{attribute addProperty BoxType "EK1100-0000-0018"}
{attribute addProperty Id "Beckhoff_EL32xxEK1122Beckhoff_EL32xxEK1122_91C4062C162A_0001_EL3201_0000_0016EL3201_E6230DF016821A_0002_EL3201_0000_0017EL3201_D2AFA85617722.125A_0003_EL3201_0000_0018EL3201_D2AFA85617722.125A_0004_EL3201_0000_0019EL3201_D2AFA85617722.125A_0005_EL3201_0000_0020EL3201_D2AFA85617722.125A_0006_EL3201_0000_0021EL3201_D2AFA85617722.125A_0007_EL3201_0000_0022EL3201_D2AFA85617722.125A_0008_EL3201_0010_0016EL3201_E6230DF016821A_0009_EL3201_0010_0017EL3201_D2AFA85617722.125A_0010_EL3201_0010_0018EL3201_D2AFA85617722.125A_0011_EL3201_0010_0019EL3201_D2AFA85617722.125A_0012_EL3201_0010_0020EL3201_D2AFA85617722.125A_0013_EL3201_0010_0021EL3201_D2AFA85617722.125A_0014_EL3201_0010_0022EL3201_D2AFA85617722.125A_0015_EL3201_0020_0016EL3201_E6230DF016821A_0016_EL3201_0020_0017EL3201_D2AFA85617722.125A_0017_EL3201_0020_0018EL3201_D2AFA85617722.125A_0018_EL3201_0020_0019EL3201_D2AFA85617722.125A_0019_EL3201_0020_0020EL3201_D2AFA85617722.125A_0020_EL3201_0020_0021EL3201_D2AFA85617722.125A_0021_EL3201_0020_0022EL3201_D2AFA85617722.125A_0022_EL3202_0000_0016EL3202_DE79C1A224030A_0023_EL3202_0000_0017EL3202_5359D6C325832.25A_0024_EL3202_0000_0018EL3202_5359D6C325832.25A_0025_EL3202_0000_0019EL3202_5359D6C325832.25A_0026_EL3202_0000_0020EL3202_5359D6C325832.25A_0027_EL3202_0000_0021EL3202_5359D6C325832.25A_0028_EL3202_0000_0022EL3202_5359D6C325832.25A_0029_EL3202_0010_0016EL3202_DE79C1A224030A_0030_EL3202_0010_0017EL3202_5359D6C325832.25A_0031_EL3202_0010_0018EL3202_5359D6C325832.25A_0032_EL3202_0010_0019EL3202_5359D6C325832.25A_0033_EL3202_0010_0020EL3202_5359D6C325832.25A_0034_EL3202_0010_0021EL3202_5359D6C325832.25A_0035_EL3202_0010_0022EL3202_5359D6C325832.25A_0036_EL3202_0020_0017EL3202_5359D6C325832.25A_0037_EL3202_0020_0018EL3202_5359D6C325832.25A_0038_EL3202_0020_0019EL3202_5359D6C325832.25A_0039_EL3202_0020_0020EL3202_5359D6C325832.25A_0040_EL3202_0020_0021EL3202_5359D6C325832.25A_0041_EL3202_0020_0022EL3202_5359D6C325832.25A_0042_EL3204_0000_0016EL3204_5D3AF62938448A_0043_EL3204_0000_0017EL3204_6E5DE15842052.5A_0044_EL3204_0000_0018EL3204_6E5DE15842052.5A_0045_EL3204_0000_0019EL3204_6E5DE15842052.5A_0046_EL3204_0000_0020EL3204_6E5DE15842052.5A_0047_EL3204_0000_0021EL3204_6E5DE15842052.5A_0048_EL3204_0162_0016EL3204_34C8240A22428A_0049_EL3204_0162_0017EL3204_34C8240A22428A_0050_EL3204_0162_0018EL3204_34C8240A22428A_0051_EL3204_0162_0019EL3204_34C8240A22428A_0052_EL3204_0200_0016EL3204_6BC1D0AA22428A_0053_EL3204_0200_0017EL3204_6BC1D0AA22428A_0054_EL3204_0200_0018EL3204_6BC1D0AA22428A_0055_EL3208_0000_0017EL3208_6C7FE11635244A_0056_EL3208_0000_0018EL3208_6C7FE11635244A_0057_EL3208_0010_0016EL3208_6C7FE11635244A_0058_EL3214_0000_0016EL3214_6BC1D0AA22428A_0059_EL3214_0000_0017EL3214_6BC1D0AA22428A_0060_EL3214_0090_0016EL3214_6BC1D0AA22428A_0061_EL3218_0000_0016EL3218_6C7FE11635244A_0062_EL3218_0000_0017EL3218_6C7FE11635244A_0063_EL3255_0000_0016EL3255_3E81353E25632A_0064_EL3255_0000_0017EL3255_0AEBB40125632A_0065_EL3255_0000_0018EL3255_0AEBB40125632A_0066_EL3255_0000_0019EL3255_0AEBB40125632A_0067_EL3255_0000_0020EL3255_2CD3FD4820826A_0068_EL3255_0000_0021EL3255_A08AFE1A25632A_0069_EL3255_0000_0022EL3255_A08AFE1A25632A_0070_EL3255_0000_0023EL3255_A08AFE1A25632"}
{attribute addProperty CRC "491847296"}
{attribute addProperty SizeInBites "17314"}
{attribute addProperty SizeInBytes "2164.25"}
TYPE Beckhoff_EL32xx_1D50FE80 EXTENDS EK1100_179A0949 :
STRUCT
	{attribute addProperty Name "Beckhoff_EL32xxEK1122"}
	Beckhoff_EL32xxEK1122 : Beckhoff_EL32xxEK1122_91C4062C;
	{attribute addProperty Name "A_0001_EL3201_0000_0016"}
	A_0001_EL3201_0000_0016 : EL3201_E6230DF0;
	{attribute addProperty Name "A_0002_EL3201_0000_0017"}
	A_0002_EL3201_0000_0017 : EL3201_D2AFA856;
	{attribute addProperty Name "A_0003_EL3201_0000_0018"}
	A_0003_EL3201_0000_0018 : EL3201_D2AFA856;
	{attribute addProperty Name "A_0004_EL3201_0000_0019"}
	A_0004_EL3201_0000_0019 : EL3201_D2AFA856;
	{attribute addProperty Name "A_0005_EL3201_0000_0020"}
	A_0005_EL3201_0000_0020 : EL3201_D2AFA856;
	{attribute addProperty Name "A_0006_EL3201_0000_0021"}
	A_0006_EL3201_0000_0021 : EL3201_D2AFA856;
	{attribute addProperty Name "A_0007_EL3201_0000_0022"}
	A_0007_EL3201_0000_0022 : EL3201_D2AFA856;
	{attribute addProperty Name "A_0008_EL3201_0010_0016"}
	A_0008_EL3201_0010_0016 : EL3201_E6230DF0;
	{attribute addProperty Name "A_0009_EL3201_0010_0017"}
	A_0009_EL3201_0010_0017 : EL3201_D2AFA856;
	{attribute addProperty Name "A_0010_EL3201_0010_0018"}
	A_0010_EL3201_0010_0018 : EL3201_D2AFA856;
	{attribute addProperty Name "A_0011_EL3201_0010_0019"}
	A_0011_EL3201_0010_0019 : EL3201_D2AFA856;
	{attribute addProperty Name "A_0012_EL3201_0010_0020"}
	A_0012_EL3201_0010_0020 : EL3201_D2AFA856;
	{attribute addProperty Name "A_0013_EL3201_0010_0021"}
	A_0013_EL3201_0010_0021 : EL3201_D2AFA856;
	{attribute addProperty Name "A_0014_EL3201_0010_0022"}
	A_0014_EL3201_0010_0022 : EL3201_D2AFA856;
	{attribute addProperty Name "A_0015_EL3201_0020_0016"}
	A_0015_EL3201_0020_0016 : EL3201_E6230DF0;
	{attribute addProperty Name "A_0016_EL3201_0020_0017"}
	A_0016_EL3201_0020_0017 : EL3201_D2AFA856;
	{attribute addProperty Name "A_0017_EL3201_0020_0018"}
	A_0017_EL3201_0020_0018 : EL3201_D2AFA856;
	{attribute addProperty Name "A_0018_EL3201_0020_0019"}
	A_0018_EL3201_0020_0019 : EL3201_D2AFA856;
	{attribute addProperty Name "A_0019_EL3201_0020_0020"}
	A_0019_EL3201_0020_0020 : EL3201_D2AFA856;
	{attribute addProperty Name "A_0020_EL3201_0020_0021"}
	A_0020_EL3201_0020_0021 : EL3201_D2AFA856;
	{attribute addProperty Name "A_0021_EL3201_0020_0022"}
	A_0021_EL3201_0020_0022 : EL3201_D2AFA856;
	{attribute addProperty Name "A_0022_EL3202_0000_0016"}
	A_0022_EL3202_0000_0016 : EL3202_DE79C1A2;
	{attribute addProperty Name "A_0023_EL3202_0000_0017"}
	A_0023_EL3202_0000_0017 : EL3202_5359D6C3;
	{attribute addProperty Name "A_0024_EL3202_0000_0018"}
	A_0024_EL3202_0000_0018 : EL3202_5359D6C3;
	{attribute addProperty Name "A_0025_EL3202_0000_0019"}
	A_0025_EL3202_0000_0019 : EL3202_5359D6C3;
	{attribute addProperty Name "A_0026_EL3202_0000_0020"}
	A_0026_EL3202_0000_0020 : EL3202_5359D6C3;
	{attribute addProperty Name "A_0027_EL3202_0000_0021"}
	A_0027_EL3202_0000_0021 : EL3202_5359D6C3;
	{attribute addProperty Name "A_0028_EL3202_0000_0022"}
	A_0028_EL3202_0000_0022 : EL3202_5359D6C3;
	{attribute addProperty Name "A_0029_EL3202_0010_0016"}
	A_0029_EL3202_0010_0016 : EL3202_DE79C1A2;
	{attribute addProperty Name "A_0030_EL3202_0010_0017"}
	A_0030_EL3202_0010_0017 : EL3202_5359D6C3;
	{attribute addProperty Name "A_0031_EL3202_0010_0018"}
	A_0031_EL3202_0010_0018 : EL3202_5359D6C3;
	{attribute addProperty Name "A_0032_EL3202_0010_0019"}
	A_0032_EL3202_0010_0019 : EL3202_5359D6C3;
	{attribute addProperty Name "A_0033_EL3202_0010_0020"}
	A_0033_EL3202_0010_0020 : EL3202_5359D6C3;
	{attribute addProperty Name "A_0034_EL3202_0010_0021"}
	A_0034_EL3202_0010_0021 : EL3202_5359D6C3;
	{attribute addProperty Name "A_0035_EL3202_0010_0022"}
	A_0035_EL3202_0010_0022 : EL3202_5359D6C3;
	{attribute addProperty Name "A_0036_EL3202_0020_0017"}
	A_0036_EL3202_0020_0017 : EL3202_5359D6C3;
	{attribute addProperty Name "A_0037_EL3202_0020_0018"}
	A_0037_EL3202_0020_0018 : EL3202_5359D6C3;
	{attribute addProperty Name "A_0038_EL3202_0020_0019"}
	A_0038_EL3202_0020_0019 : EL3202_5359D6C3;
	{attribute addProperty Name "A_0039_EL3202_0020_0020"}
	A_0039_EL3202_0020_0020 : EL3202_5359D6C3;
	{attribute addProperty Name "A_0040_EL3202_0020_0021"}
	A_0040_EL3202_0020_0021 : EL3202_5359D6C3;
	{attribute addProperty Name "A_0041_EL3202_0020_0022"}
	A_0041_EL3202_0020_0022 : EL3202_5359D6C3;
	{attribute addProperty Name "A_0042_EL3204_0000_0016"}
	A_0042_EL3204_0000_0016 : EL3204_5D3AF629;
	{attribute addProperty Name "A_0043_EL3204_0000_0017"}
	A_0043_EL3204_0000_0017 : EL3204_6E5DE158;
	{attribute addProperty Name "A_0044_EL3204_0000_0018"}
	A_0044_EL3204_0000_0018 : EL3204_6E5DE158;
	{attribute addProperty Name "A_0045_EL3204_0000_0019"}
	A_0045_EL3204_0000_0019 : EL3204_6E5DE158;
	{attribute addProperty Name "A_0046_EL3204_0000_0020"}
	A_0046_EL3204_0000_0020 : EL3204_6E5DE158;
	{attribute addProperty Name "A_0047_EL3204_0000_0021"}
	A_0047_EL3204_0000_0021 : EL3204_6E5DE158;
	{attribute addProperty Name "A_0048_EL3204_0162_0016"}
	A_0048_EL3204_0162_0016 : EL3204_34C8240A;
	{attribute addProperty Name "A_0049_EL3204_0162_0017"}
	A_0049_EL3204_0162_0017 : EL3204_34C8240A;
	{attribute addProperty Name "A_0050_EL3204_0162_0018"}
	A_0050_EL3204_0162_0018 : EL3204_34C8240A;
	{attribute addProperty Name "A_0051_EL3204_0162_0019"}
	A_0051_EL3204_0162_0019 : EL3204_34C8240A;
	{attribute addProperty Name "A_0052_EL3204_0200_0016"}
	A_0052_EL3204_0200_0016 : EL3204_6BC1D0AA;
	{attribute addProperty Name "A_0053_EL3204_0200_0017"}
	A_0053_EL3204_0200_0017 : EL3204_6BC1D0AA;
	{attribute addProperty Name "A_0054_EL3204_0200_0018"}
	A_0054_EL3204_0200_0018 : EL3204_6BC1D0AA;
	{attribute addProperty Name "A_0055_EL3208_0000_0017"}
	A_0055_EL3208_0000_0017 : EL3208_6C7FE116;
	{attribute addProperty Name "A_0056_EL3208_0000_0018"}
	A_0056_EL3208_0000_0018 : EL3208_6C7FE116;
	{attribute addProperty Name "A_0057_EL3208_0010_0016"}
	A_0057_EL3208_0010_0016 : EL3208_6C7FE116;
	{attribute addProperty Name "A_0058_EL3214_0000_0016"}
	A_0058_EL3214_0000_0016 : EL3214_6BC1D0AA;
	{attribute addProperty Name "A_0059_EL3214_0000_0017"}
	A_0059_EL3214_0000_0017 : EL3214_6BC1D0AA;
	{attribute addProperty Name "A_0060_EL3214_0090_0016"}
	A_0060_EL3214_0090_0016 : EL3214_6BC1D0AA;
	{attribute addProperty Name "A_0061_EL3218_0000_0016"}
	A_0061_EL3218_0000_0016 : EL3218_6C7FE116;
	{attribute addProperty Name "A_0062_EL3218_0000_0017"}
	A_0062_EL3218_0000_0017 : EL3218_6C7FE116;
	{attribute addProperty Name "A_0063_EL3255_0000_0016"}
	A_0063_EL3255_0000_0016 : EL3255_3E81353E;
	{attribute addProperty Name "A_0064_EL3255_0000_0017"}
	A_0064_EL3255_0000_0017 : EL3255_0AEBB401;
	{attribute addProperty Name "A_0065_EL3255_0000_0018"}
	A_0065_EL3255_0000_0018 : EL3255_0AEBB401;
	{attribute addProperty Name "A_0066_EL3255_0000_0019"}
	A_0066_EL3255_0000_0019 : EL3255_0AEBB401;
	{attribute addProperty Name "A_0067_EL3255_0000_0020"}
	A_0067_EL3255_0000_0020 : EL3255_2CD3FD48;
	{attribute addProperty Name "A_0068_EL3255_0000_0021"}
	A_0068_EL3255_0000_0021 : EL3255_A08AFE1A;
	{attribute addProperty Name "A_0069_EL3255_0000_0022"}
	A_0069_EL3255_0000_0022 : EL3255_A08AFE1A;
	{attribute addProperty Name "A_0070_EL3255_0000_0023"}
	A_0070_EL3255_0000_0023 : EL3255_A08AFE1A;
END_STRUCT
END_TYPE

(* stored: Version 1.2.0.0, ProductVersion 3.1.4024.9
   DUT Beckhoff_EL32xx_1D50FE80: Id {9ccd6757-67d6-42e7-aa73-2760df15ecf3} *)
